TYPE ST_IO2_SingleInputLockedCtrl :
STRUCT
	eTypeInput 		: E_IO2_Type;
	tTimeOnFilter		: TIME;
	tTimeOffFilter 		: TIME;
	tTimeLatch			: TIME;
	sInputName		: STRING(40);
END_STRUCT
END_TYPE

(* stored: Version 1.1.0.1
   DUT ST_IO2_SingleInputLockedCtrl: Id {a71b47ba-4c40-448d-bb2f-2bcf11fd6e13} *)
